// TIA Portal V20 export
TYPE "typeSideTapeIdleTimeHmiInterface"
// stored: Access Published, Namespace Unit1.Em4
   STRUCT
      currentCount : Time;
      processCount : Time := T#0ms;
   END_STRUCT;
END_TYPE
